FUNCTION_BLOCK WORKERA1FB (* JADE WORKER *)
  (* Standard: 61499-1 *)
  (* Version 1.0, 2014-04-22, Ahmed, Fraunhofer IGD *)
  (* Compiler header: package fb.rt; *)
  (* Compiler Java Sun JDK 1.5.0 *)
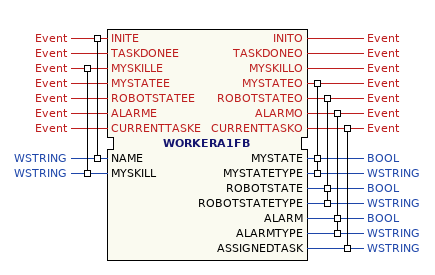
  EVENT_INPUT
    INITE WITH NAME;
    TASKDONEE;
    MYSKILLE WITH MYSKILL;
    MYSTATEE;
    ROBOTSTATEE;
    ALARME;
    CURRENTTASKE;
  END_EVENT
  EVENT_OUTPUT
    INITO;
    TASKDONEO;
    MYSKILLO;
    MYSTATEO WITH MYSTATE, MYSTATETYPE;
    ROBOTSTATEO WITH ROBOTSTATE, ROBOTSTATETYPE;
    ALARMO WITH ALARM, ALARMTYPE;
    CURRENTTASKO WITH ASSIGNEDTASK;
  END_EVENT
  VAR_INPUT
    NAME : WSTRING;
    MYSKILL : WSTRING;
  END_VAR
  VAR_OUTPUT
    MYSTATE : BOOL;
    MYSTATETYPE : WSTRING;
    ROBOTSTATE : BOOL;
    ROBOTSTATETYPE : WSTRING;
    ALARM : BOOL;
    ALARMTYPE : WSTRING;
    ASSIGNEDTASK : WSTRING;
  END_VAR
END_FUNCTION_BLOCK
